SUBAPPLICATION mapping (* Subapplication Type *)
  (* Standard: 61499-2 *)
  (* Version 1.0, 2023-10-23, franz *)
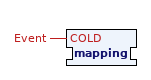
  EVENT_INPUT
    COLD;
  END_EVENT
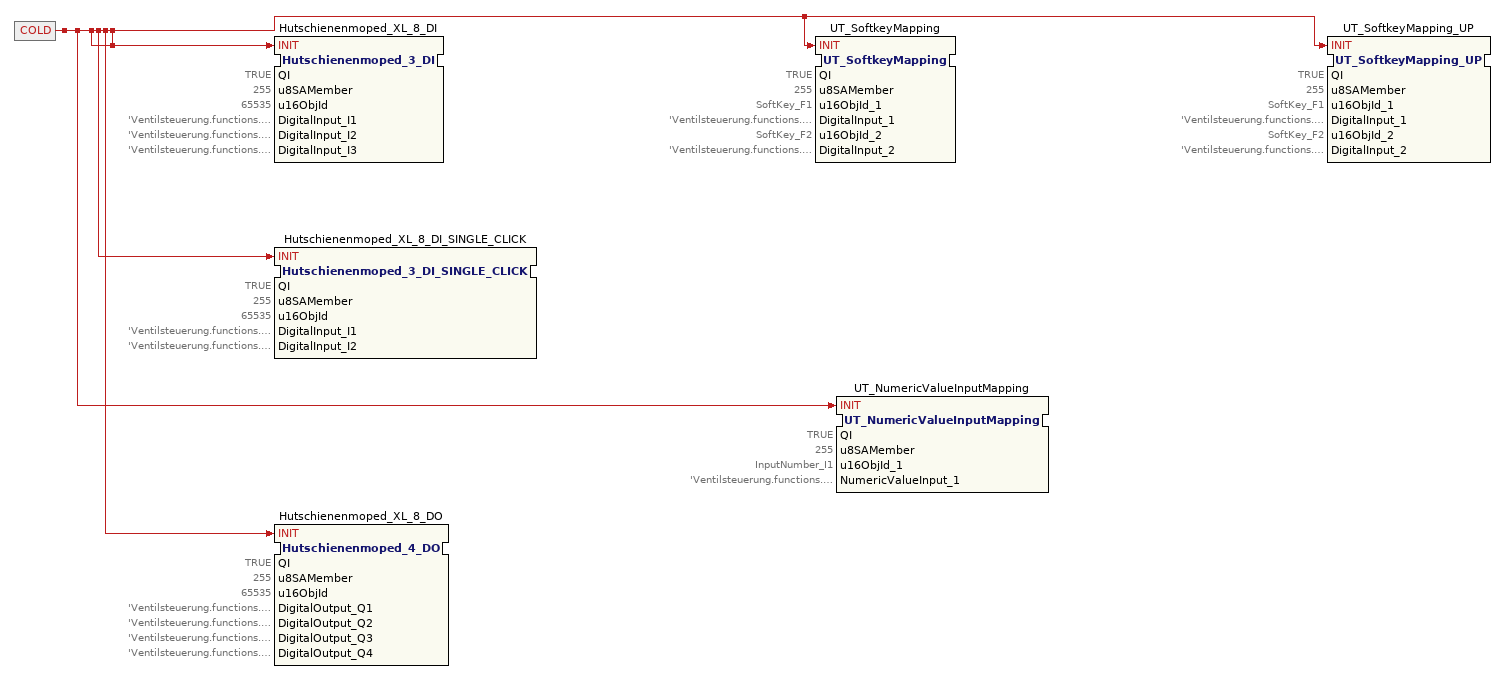
  FBS
    UT_SoftkeyMapping : UT_SoftkeyMapping(QI := TRUE, u8SAMember := 255, u16ObjId_1 := SoftKey_F1, DigitalInput_1 := 'Ventilsteuerung.functions.SoftKey_F1', u16ObjId_2 := SoftKey_F2, DigitalInput_2 := 'Ventilsteuerung.functions.SoftKey_F2');
    UT_NumericValueInputMapping : UT_NumericValueInputMapping(QI := TRUE, u8SAMember := 255, u16ObjId_1 := InputNumber_I1, NumericValueInput_1 := 'Ventilsteuerung.functions.InputNumber_I1');
    UT_SoftkeyMapping_UP : UT_SoftkeyMapping_UP(QI := TRUE, u8SAMember := 255, u16ObjId_1 := SoftKey_F1, DigitalInput_1 := 'Ventilsteuerung.functions.SoftKey_F1_UP', u16ObjId_2 := SoftKey_F2, DigitalInput_2 := 'Ventilsteuerung.functions.SoftKey_F2_UP');
    Hutschienenmoped_XL_8_DI : Hutschienenmoped_3_DI(QI := TRUE, u8SAMember := 255, u16ObjId := 65535, DigitalInput_I1 := 'Ventilsteuerung.functions.DigitalInput_I1', DigitalInput_I2 := 'Ventilsteuerung.functions.DigitalInput_I2', DigitalInput_I3 := 'Ventilsteuerung.functions.DigitalInput_I3');
    Hutschienenmoped_XL_8_DI_SINGLE_CLICK : Hutschienenmoped_3_DI_SINGLE_CLICK(QI := TRUE, u8SAMember := 255, u16ObjId := 65535, DigitalInput_I1 := 'Ventilsteuerung.functions.DigitalInput_I1_CLK', DigitalInput_I2 := 'Ventilsteuerung.functions.DigitalInput_I2_CLK');
    Hutschienenmoped_XL_8_DO : Hutschienenmoped_4_DO(QI := TRUE, u8SAMember := 255, u16ObjId := 65535, DigitalOutput_Q1 := 'Ventilsteuerung.functions.DigitalOutput_Q1', DigitalOutput_Q2 := 'Ventilsteuerung.functions.DigitalOutput_Q2', DigitalOutput_Q3 := 'Ventilsteuerung.functions.DigitalOutput_Q3', DigitalOutput_Q4 := 'Ventilsteuerung.functions.DigitalOutput_Q4');
  END_FBS
  EVENT_CONNECTIONS
    COLD TO UT_SoftkeyMapping.INIT;
    COLD TO UT_NumericValueInputMapping.INIT;
    COLD TO UT_SoftkeyMapping_UP.INIT;
    COLD TO Hutschienenmoped_XL_8_DI.INIT;
    COLD TO Hutschienenmoped_XL_8_DI_SINGLE_CLICK.INIT;
    COLD TO Hutschienenmoped_XL_8_DO.INIT;
    COLD TO Hutschienenmoped_XL_8_DI.INIT;
  END_CONNECTIONS
END_SUBAPPLICATION
